//==================================================================================================
//								RJM Maszyny sp. z o.o.
//									13.05.2022
//
//	Obsługa przycisku niepodświetlanego
//	v1.0	|| TC v 3.1.4024.22		|| - pierwsza wersja
//==================================================================================================
FUNCTION_BLOCK FB_Przycisk_NC IMPLEMENTS I_Przycisk
VAR
	Wejscie							AT %I*	: BOOL;
END_VAR

//==================================================================================================
//								RJM Maszyny sp. z o.o.
//									13.05.2022
//
//	Sprawdzenie czy wciśnięty
//	v1.0	|| TC v 3.1.4024.22		|| - pierwsza wersja
//==================================================================================================
PROPERTY CzyNacisniety : BOOL
GET
CzyNacisniety 								:= NOT Wejscie;
END_GET
END_PROPERTY

//==================================================================================================
//								RJM Maszyny sp. z o.o.
//									13.05.2022
//
//	Sprawdzenie czy puszczony
//	v1.0	|| TC v 3.1.4024.22		|| - pierwsza wersja
//==================================================================================================
PROPERTY CzyPuszczony : BOOL
GET
CzyPuszczony								:= Wejscie;
END_GET
END_PROPERTY

END_FUNCTION_BLOCK

(* stored: Version 1.1.0.1, ProductVersion 3.1.4024.11
   POU FB_Przycisk_NC: Id {0a2e6707-b6ba-4532-b715-3ce0575852b8}, SpecialFunc None
   Property CzyNacisniety: Id {412cd168-da5b-42a0-9d51-406d29cced53}
   Get Get: Id {e466453b-095a-4ec5-bcb1-02e33e2bb676}
   Property CzyPuszczony: Id {92ba1473-418b-48ae-9edf-043537775f6b}
   Get Get: Id {8f03c4b3-198f-46e5-879c-e332a08a01c4} *)
